(* Logix 5000 project; controller pracainz_ne 1769-L16ER-BB1B rev 30.11; software revision 30.00; part 2 of 2 *)
(* tags used below, declared in another part *)
   BELT_CONV_2_0 : ALIAS FOR BOOL_OUT_0;
   BELT_CONV_2_1 : ALIAS FOR BOOL_OUT_1;
   BELT_CONV_2_2 : ALIAS FOR BOOL_OUT_2;
   BELT_CONV_2_3 : ALIAS FOR BOOL_OUT_3;
   BELT_CONV_2_4 : ALIAS FOR BOOL_OUT_4;
   BELT_CONV_2_5 : ALIAS FOR BOOL_OUT_5;
   BELT_CONV_2_6 : ALIAS FOR BOOL_OUT_6;
   BELT_CONV_2_7 : ALIAS FOR BOOL_OUT_7;
   BELT_CONV_2_CCW : ALIAS FOR BOOL_OUT_27;
   BELT_CONV_4_0 : ALIAS FOR BOOL_OUT_8;
   BELT_CONV_4_1 : ALIAS FOR BOOL_OUT_9;
   BELT_CONV_4_2 : ALIAS FOR BOOL_OUT_10;
   BELT_CONV_4_3 : ALIAS FOR BOOL_OUT_11;
   BELT_CONV_CCW_0 : ALIAS FOR BOOL_OUT_23;
   BELT_CONV_CCW_3 : ALIAS FOR BOOL_OUT_24;
   BELT_CONV_CCW_4 : ALIAS FOR BOOL_OUT_25;
   BELT_CONV_CW_0 : ALIAS FOR BOOL_OUT_26;
   BELT_CONV_CW_1 : ALIAS FOR BOOL_OUT_20;
   BELT_CONV_CW_2 : ALIAS FOR BOOL_OUT_21;
   BELT_CONV_CW_5 : ALIAS FOR BOOL_OUT_22;
   CAP_SEN_0 : ALIAS FOR BOOL_IN_0;
   CAP_SEN_1 : ALIAS FOR BOOL_IN_1;
   CHAIN_0_LEFT : ALIAS FOR BOOL_OUT_16;
   CHAIN_0_N : ALIAS FOR BOOL_OUT_13;
   CHAIN_0_P : ALIAS FOR BOOL_OUT_12;
   CHAIN_0_RIGHT : ALIAS FOR BOOL_OUT_18;
   CHAIN_1_LEFT : ALIAS FOR BOOL_OUT_17;
   CHAIN_1_N : ALIAS FOR BOOL_OUT_15;
   CHAIN_1_P : ALIAS FOR BOOL_OUT_14;
   CHAIN_1_RIGHT : ALIAS FOR BOOL_OUT_19;
   COUNT : DINT;
   DIFF_SEN_0 : ALIAS FOR BOOL_IN_4;
   DIFF_SEN_1 : ALIAS FOR BOOL_IN_5;
   DIFF_SEN_2 : ALIAS FOR BOOL_IN_6;
   MANUAL : ALIAS FOR M_04;
   NOT_BLUE : ALIAS FOR M_24;
   NOT_GREEN : ALIAS FOR M_23;
   OSF_08_O : ALIAS FOR M_41;
   OSF_08_S : ALIAS FOR M_42;
   OSR_06_O : ALIAS FOR M_33;
   OSR_06_S : ALIAS FOR M_34;
   OSR_07_O : ALIAS FOR M_35;
   OSR_07_S : ALIAS FOR M_36;
   P_P_0_DETE : ALIAS FOR BOOL_IN_20;
   P_P_0_GRAB : ALIAS FOR BOOL_OUT_45;
   P_P_0_X : ALIAS FOR FLOAT_OUT_2;
   P_P_0_X_POSITION : ALIAS FOR FLOAT_IN_1;
   P_P_0_Y : ALIAS FOR FLOAT_OUT_0;
   P_P_0_Y_POSITION : ALIAS FOR FLOAT_IN_2;
   P_P_0_Z : ALIAS FOR FLOAT_OUT_4;
   P_P_0_Z_POSITION : ALIAS FOR FLOAT_IN_3;
   P_P_1_DETE : ALIAS FOR BOOL_IN_21;
   P_P_1_GRAB : ALIAS FOR BOOL_OUT_46;
   P_P_1_X : ALIAS FOR FLOAT_OUT_3;
   P_P_1_X_D : REAL;
   P_P_1_X_POSITION : ALIAS FOR FLOAT_IN_4;
   P_P_1_Y : ALIAS FOR FLOAT_OUT_1;
   P_P_1_Y_D : REAL;
   P_P_1_Y_POSITION : ALIAS FOR FLOAT_IN_5;
   P_P_1_Z : ALIAS FOR FLOAT_OUT_5;
   P_P_1_Z_D : REAL;
   P_P_1_Z_POSITION : ALIAS FOR FLOAT_IN_6;
   PUSH_0 : ALIAS FOR BOOL_OUT_47;
   PUSH_1 : ALIAS FOR BOOL_OUT_48;
   PUSHER_1 : BOOL;
   RETRO_SEN_0 : ALIAS FOR BOOL_IN_25;
   RETRO_SEN_3 : ALIAS FOR BOOL_IN_28;
   ROLL_4_0 : ALIAS FOR BOOL_OUT_50;
   ROLL_4_1 : ALIAS FOR BOOL_OUT_51;
   ROLL_4_2 : ALIAS FOR BOOL_OUT_52;
   ROLL_6_0 : ALIAS FOR BOOL_OUT_53;
   ROLL_6_1 : ALIAS FOR BOOL_OUT_54;
   TASMA_1 : BOOL;
   TASMA_2 : BOOL;
   TASMA_5 : BOOL;
   TASMA_9 : BOOL;
   auto_once : BOOL;
   BOOL_IN_41 : BOOL;
   BOOL_IN_43 : BOOL;
   BOOL_OUT_0 : BOOL;
   BOOL_OUT_1 : BOOL;
   BOOL_OUT_10 : BOOL;
   BOOL_OUT_11 : BOOL;
   BOOL_OUT_12 : BOOL;
   BOOL_OUT_13 : BOOL;
   BOOL_OUT_14 : BOOL;
   BOOL_OUT_15 : BOOL;
   BOOL_OUT_16 : BOOL;
   BOOL_OUT_17 : BOOL;
   BOOL_OUT_18 : BOOL;
   BOOL_OUT_19 : BOOL;
   BOOL_OUT_2 : BOOL;
   BOOL_OUT_20 : BOOL;
   BOOL_OUT_21 : BOOL;
   BOOL_OUT_22 : BOOL;
   BOOL_OUT_23 : BOOL;
   BOOL_OUT_24 : BOOL;
   BOOL_OUT_25 : BOOL;
   BOOL_OUT_26 : BOOL;
   BOOL_OUT_27 : BOOL;
   BOOL_OUT_29 : BOOL;
   BOOL_OUT_3 : BOOL;
   BOOL_OUT_30 : BOOL;
   BOOL_OUT_32 : BOOL;
   BOOL_OUT_33 : BOOL;
   BOOL_OUT_34 : BOOL;
   BOOL_OUT_35 : BOOL;
   BOOL_OUT_36 : BOOL;
   BOOL_OUT_37 : BOOL;
   BOOL_OUT_38 : BOOL;
   BOOL_OUT_39 : BOOL;
   BOOL_OUT_4 : BOOL;
   BOOL_OUT_40 : BOOL;
   BOOL_OUT_41 : BOOL;
   BOOL_OUT_42 : BOOL;
   BOOL_OUT_43 : BOOL;
   BOOL_OUT_44 : BOOL;
   BOOL_OUT_45 : BOOL;
   BOOL_OUT_46 : BOOL;
   BOOL_OUT_47 : BOOL;
   BOOL_OUT_48 : BOOL;
   BOOL_OUT_5 : BOOL;
   BOOL_OUT_50 : BOOL;
   BOOL_OUT_51 : BOOL;
   BOOL_OUT_52 : BOOL;
   BOOL_OUT_53 : BOOL;
   BOOL_OUT_54 : BOOL;
   BOOL_OUT_55 : BOOL;
   BOOL_OUT_56 : BOOL;
   BOOL_OUT_57 : BOOL;
   BOOL_OUT_6 : BOOL;
   BOOL_OUT_7 : BOOL;
   BOOL_OUT_8 : BOOL;
   BOOL_OUT_9 : BOOL;
   CHAIN_1_B : BOOL;
   CHAIN_1_F : BOOL;
   CHAIN_1_L : BOOL;
   CHAIN_1_R : BOOL;
   CHAIN_2_B : BOOL;
   CHAIN_2_F : BOOL;
   CHAIN_2_L : BOOL;
   CHAIN_2_R : BOOL;
   CLAMPED : BOOL;
   CLAMPED_R : BOOL;
   COUNT_R : DINT;
   EMERGENCY_ALL : BOOL;
   END_OF_DAY : BOOL;
   full_palet : BOOL;
   FULL_PALET_R : BOOL;
   Input_1 : BOOL;
   Input_1_R : BOOL;
   Input_2 : BOOL;
   Input_2_R : BOOL;
   Input_3 : BOOL;
   Input_3_R : BOOL;
   Input_4 : BOOL;
   Input_4_R : BOOL;
   Input_5 : BOOL;
   Input_5_R : BOOL;
   Input_6 : BOOL;
   Input_6_R : BOOL;
   Input_7 : BOOL;
   Input_7_R : BOOL;
   LEFT_PACK : BOOL;
   LEFT_PICK : BOOL;
   LEWA_LINIA : BOOL;
   LEWA_STRONA : BOOL;
   manual_once : BOOL;
   OSR_10_O : BOOL;
   OSR_10_S : BOOL;
   OSR_13_O : BOOL;
   OSR_14_O : BOOL;
   OSR_14_S : BOOL;
   P_P_0_X_D : REAL;
   P_P_0_Y_D : REAL;
   P_P_0_Z_D : REAL;
   PICK : BOOL;
   PRAWA_LINIA : BOOL;
   PRAWA_STRONA : BOOL;
   PUSHER_2 : BOOL;
   READY_L : BOOL;
   READY_R : BOOL;
   reset_timer : BOOL;
   reset_timer_l : BOOL;
   RIGHT_PACK : BOOL;
   RIGHT_PICK : BOOL;
   ROLL_1 : BOOL;
   ROLL_2 : BOOL;
   ROLL_3 : BOOL;
   ROLL_4 : BOOL;
   ROLL_5 : BOOL;
   ROLL_6 : BOOL;
   ROLL_7 : BOOL;
   START_ALL : BOOL;
   STOP_LEFT : BOOL;
   STOP_RIGHT : BOOL;
   stopped_left : BOOL;
   stopped_right : BOOL;
   TASMA_1_P : BOOL;
   TASMA_2_P : BOOL;
   TASMA_5_P : BOOL;
   TASMA_9_P : BOOL;
   TIMER_LEFT_P_P : TIMER;
   TIMER_RIGHT_P_P : TIMER;
   ton1 : TIMER;
   TON1_R : TIMER;
   ton2 : TIMER;
   TON2_R : TIMER;
   ton3 : TIMER;
   ton3_R : TIMER;
   ton4 : TIMER;
   TON4_R : TIMER;
   ton5 : TIMER;
   TON5_R : TIMER;
   ton6 : TIMER;
   TON6_R : TIMER;
   TON7 : TIMER;
   TON7_R : TIMER;
   X0 : REAL;
   X1 : REAL;
   Y0 : REAL;
   Y1 : REAL;
(* MainProgram, continued *)

ROUTINE R_07_timer_PICKNPLACE   (* ladder *)
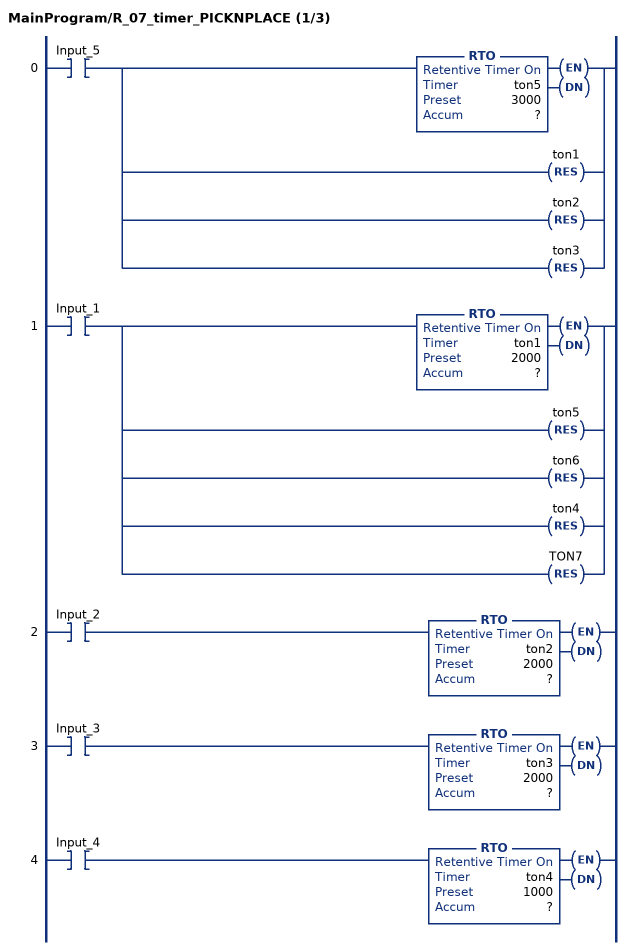
   0: XIC(Input_5)[RTO(ton5,?,?) ,RES(ton1) ,RES(ton2) ,RES(ton3) ];
   1: XIC(Input_1)[RTO(ton1,?,?) ,RES(ton5) ,RES(ton6) ,RES(ton4) ,RES(TON7) ];
   2: XIC(Input_2)RTO(ton2,?,?);
   3: XIC(Input_3)RTO(ton3,?,?);
   4: XIC(Input_4)RTO(ton4,?,?);
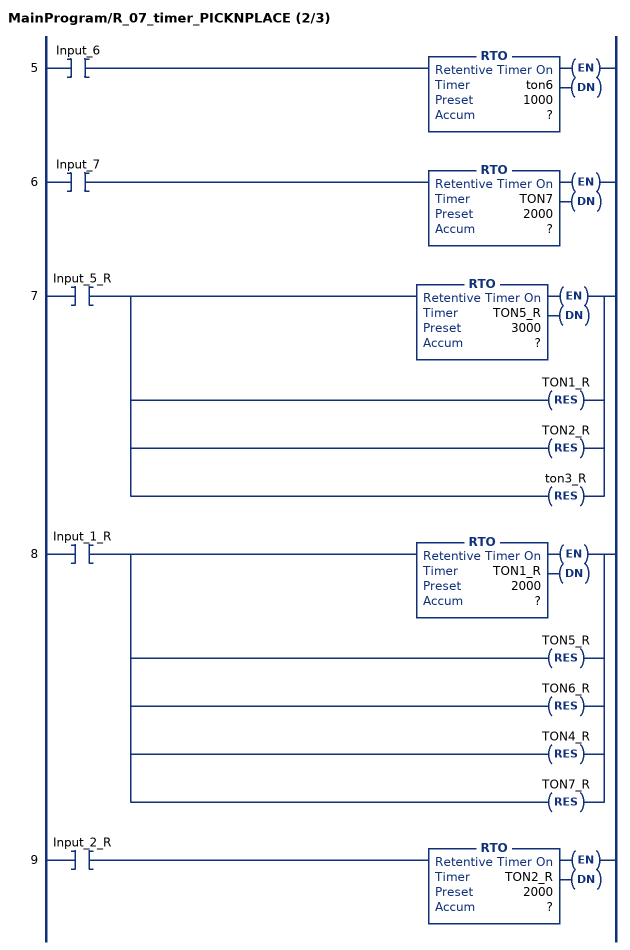
   5: XIC(Input_6)RTO(ton6,?,?);
   6: XIC(Input_7)RTO(TON7,?,?);
   7: XIC(Input_5_R)[RTO(TON5_R,?,?) ,RES(TON1_R) ,RES(TON2_R) ,RES(ton3_R) ];
   8: XIC(Input_1_R)[RTO(TON1_R,?,?) ,RES(TON5_R) ,RES(TON6_R) ,RES(TON4_R) ,RES(TON7_R) ];
   9: XIC(Input_2_R)RTO(TON2_R,?,?);
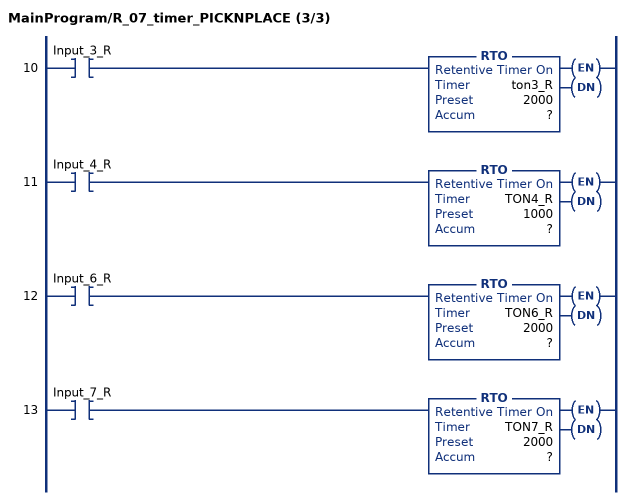
   10: XIC(Input_3_R)RTO(ton3_R,?,?);
   11: XIC(Input_4_R)RTO(TON4_R,?,?);
   12: XIC(Input_6_R)RTO(TON6_R,?,?);
   13: XIC(Input_7_R)RTO(TON7_R,?,?);
END_ROUTINE

ROUTINE R_08_Pick_and_Place_L   (* structured text *)
   IF LEFT_PACK THEN
   LEFT_PICK:=1;
   Input_1:=0;
   Input_2:=0;
   Input_3:=0;
   END_IF;
   
   IF  LEFT_PICK AND NOT(BOOL_IN_43) AND NOT(CLAMPED) AND (TIMER_LEFT_P_P.DN ) THEN  // ZACISKANIE
   BOOL_OUT_57:=1;
   END_IF;
   
   IF BOOL_IN_43 THEN
   CLAMPED:=1;
   BOOL_OUT_57:=0;
   P_P_1_Z:=0;
   Input_5:=1;
   END_IF;
   
   IF  LEFT_PICK AND CLAMPED THEN  // ZACZYNAMY OPERACJE RAMIENIEM
   LEFT_PICK:=0;
   END_IF;
   
   IF (Input_5)  THEN  // CHWYTANIE
   P_P_1_X:=9.1;
   P_P_1_Y:=6.5;
   IF ((P_P_1_X_POSITION=9.1) AND (P_P_1_Y_POSITION=6.5)) OR ton5.DN THEN
   P_P_1_Z:=8.5;
   IF (P_P_1_Z_POSITION>8.49 AND CLAMPED) then
   IF(P_P_1_DETE)THEN
   P_P_1_GRAB:=1;
   Input_6:=1;
   ELSE
   reset_timer_l:=1;
   CLAMPED:=0;
   END_IF;
   END_IF;
   END_IF;
   END_IF;
   
   
   IF  ton6.DN THEN
   P_P_1_Z:=0;
   Input_4:=1;
   IF ton4.DN THEN
   COUNT:=COUNT+1;
   READY_L:=1;
   LEFT_PICK:=0;
   END_IF;
   END_IF;
   
   
   
   
   IF READY_L AND NOT(full_palet) AND NOT(RETRO_SEN_0)  THEN
   
   CLAMPED:=0;
   Input_4:=0;
   Input_5:=0;
   Input_6:=0;
   Input_7:=0;
   
   CASE COUNT OF
   1:
   X1:=3.5;
   Y1:=6.8;
   
   2:
   X1:=5.29;
   Y1:=6.8;
   
   3:
   X1:=3.5;
   Y1:=3.8;
   
   4:
   X1:=5.29;
   Y1:=3.8;
   END_CASE;
   
   Input_1:=1;
   P_P_1_X:=X1;
   P_P_1_Y:=Y1;
   IF ((P_P_1_X_POSITION=X1) AND (P_P_1_Y_POSITION=Y1)) OR ton1.DN THEN
   P_P_1_Z:=8.5;
   Input_2:=1;
   IF (P_P_1_Z_POSITION>8.49) AND ton2.DN THEN
   P_P_1_GRAB:=0;
   P_P_1_Z:=5;
   READY_L:=0;
   END_IF;
   END_IF;
   END_IF;
   
   IF(COUNT=4) AND NOT(P_P_1_GRAB) THEN
   full_palet:=1;
   COUNT:=0;
   
   END_IF;
   
   
   
END_ROUTINE

ROUTINE R_08_Pick_and_Place_R   (* structured text *)
   IF RIGHT_PACK THEN
   RIGHT_PICK:=1;
   Input_1_R:=0;
   Input_2_R:=0;
   Input_3_R:=0;
   
   END_IF;
   
   IF  RIGHT_PICK AND NOT(BOOL_IN_41) AND NOT(CLAMPED_R) AND (TIMER_RIGHT_P_P.DN) THEN  // ZACISKANIE
   BOOL_OUT_55:=1;
   END_IF;
   
   IF BOOL_IN_41 THEN
   CLAMPED_R:=1;
   BOOL_OUT_55:=0;
   P_P_0_Z:=0;
   Input_5_R:=1;
   END_IF;
   
   IF  RIGHT_PICK AND CLAMPED_R THEN  // ZACZYNAMY OPERACJE RAMIENIEM
   RIGHT_PICK:=0;
   END_IF;
   
   IF (Input_5_R)  THEN  // CHWYTANIE
   P_P_0_X:=9.1;
   P_P_0_Y:=6.5;
   IF ((P_P_0_X_POSITION=9.1) AND (P_P_0_Y_POSITION=6.5)) OR TON5_R.DN THEN
   P_P_0_Z:=8.5;
   Input_7_R:=1;
   IF (P_P_0_Z_POSITION>8.49 AND CLAMPED_R) THEN
   IF(P_P_0_DETE)and TON7_R.DN THEN
   P_P_0_GRAB:=1;
   Input_6_R:=1;
   else
   reset_timer:=1;
   CLAMPED_R:=0;
   END_IF;
   END_IF;
   END_IF;
   END_IF;
   
   
   
   IF  TON6_R.DN THEN
   P_P_0_Z:=0;
   Input_4_R:=1;
   IF TON4_R.DN THEN
   COUNT_R:=COUNT_R+1;
   READY_R:=1;
   RIGHT_PICK:=0;
   END_IF;
   END_IF;
   
   
   
   IF READY_R AND NOT(FULL_PALET_R) AND NOT(RETRO_SEN_3)  THEN
   CLAMPED_R:=0;
   Input_4_R:=0;
   Input_5_R:=0;
   Input_6_R:=0;
   Input_7_R:=0;
   
   CASE COUNT_R OF
   1:
   X0:=3.5;
   Y0:=6.0;
   
   2:
   X0:=5.3;
   Y0:=6.0;
   
   3:
   X0:=3.5;
   Y0:=2.9;
   
   4:
   X0:=5.3;
   Y0:=2.9;
   END_CASE;
   
   Input_1_R:=1;
   P_P_0_X:=X0;
   P_P_0_Y:=Y0;
   IF ((P_P_0_X_POSITION=X0) AND (P_P_0_Y_POSITION=Y0)) OR TON1_R.DN THEN
   P_P_0_Z:=8.5;
   Input_2_R:=1;
   IF (P_P_0_Z_POSITION>8.49) AND TON2_R.DN THEN
   P_P_0_GRAB:=0;
   P_P_0_Z:=5;
   READY_R:=0;
   END_IF;
   END_IF;
   END_IF;
   
   IF(COUNT_R=4) AND NOT(P_P_0_GRAB) THEN
   FULL_PALET_R:=1;
   COUNT_R:=0;
   
   END_IF;
   
   
   
END_ROUTINE

ROUTINE R_09_roller_n_chain   (* ladder *)
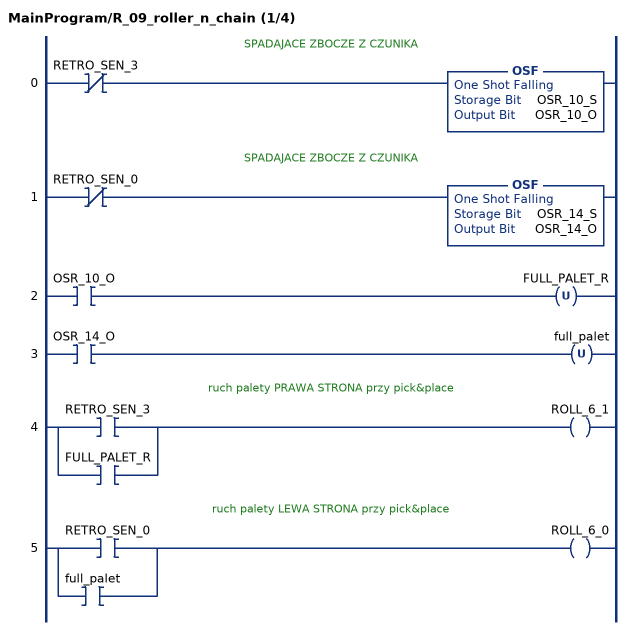
   // SPADAJACE ZBOCZE Z CZUNIKA
   0: XIO(RETRO_SEN_3)OSF(OSR_10_S,OSR_10_O);
   // SPADAJACE ZBOCZE Z CZUNIKA
   1: XIO(RETRO_SEN_0)OSF(OSR_14_S,OSR_14_O);
   2: XIC(OSR_10_O)OTU(FULL_PALET_R);
   3: XIC(OSR_14_O)OTU(full_palet);
   // ruch palety PRAWA STRONA przy pick&place
   4: [XIC(RETRO_SEN_3) ,XIC(FULL_PALET_R) ]OTE(ROLL_6_1);
   // ruch palety LEWA STRONA przy pick&place
   5: [XIC(RETRO_SEN_0) ,XIC(full_palet) ]OTE(ROLL_6_0);
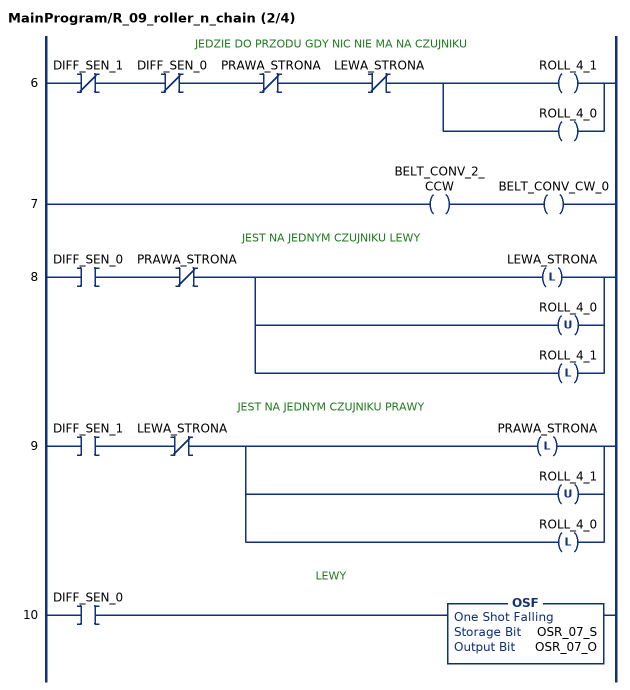
   // JEDZIE DO PRZODU GDY NIC NIE MA NA CZUJNIKU
   6: XIO(DIFF_SEN_1)XIO(DIFF_SEN_0)XIO(PRAWA_STRONA)XIO(LEWA_STRONA)[OTE(ROLL_4_1) ,OTE(ROLL_4_0) ];
   7: OTE(BELT_CONV_2_CCW)OTE(BELT_CONV_CW_0);
   // JEST NA JEDNYM CZUJNIKU LEWY
   8: XIC(DIFF_SEN_0)XIO(PRAWA_STRONA)[OTL(LEWA_STRONA) ,OTU(ROLL_4_0) ,OTL(ROLL_4_1) ];
   // JEST NA JEDNYM CZUJNIKU PRAWY
   9: XIC(DIFF_SEN_1)XIO(LEWA_STRONA)[OTL(PRAWA_STRONA) ,OTU(ROLL_4_1) ,OTL(ROLL_4_0) ];
   // LEWY
   10: XIC(DIFF_SEN_0)OSF(OSR_07_S,OSR_07_O);
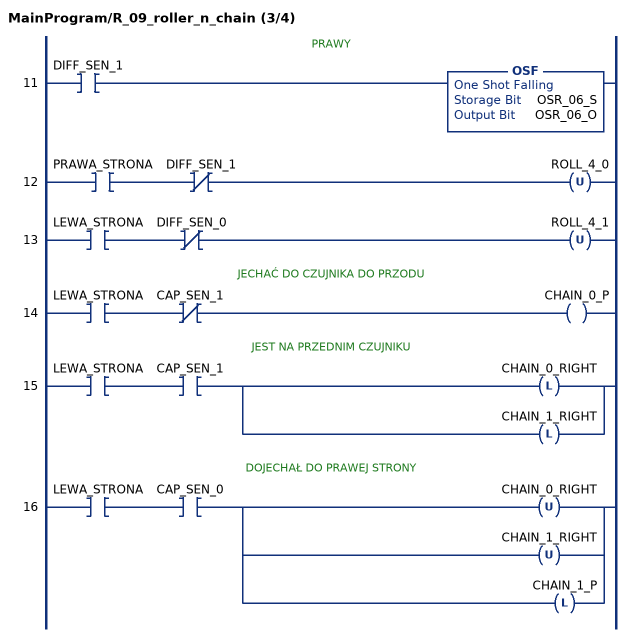
   // PRAWY
   11: XIC(DIFF_SEN_1)OSF(OSR_06_S,OSR_06_O);
   12: XIC(PRAWA_STRONA)XIO(DIFF_SEN_1)OTU(ROLL_4_0);
   13: XIC(LEWA_STRONA)XIO(DIFF_SEN_0)OTU(ROLL_4_1);
   // JECHAĆ DO CZUJNIKA DO PRZODU
   14: XIC(LEWA_STRONA)XIO(CAP_SEN_1)OTE(CHAIN_0_P);
   // JEST NA PRZEDNIM CZUJNIKU
   15: XIC(LEWA_STRONA)XIC(CAP_SEN_1)[OTL(CHAIN_0_RIGHT) ,OTL(CHAIN_1_RIGHT) ];
   // DOJECHAŁ DO PRAWEJ STRONY
   16: XIC(LEWA_STRONA)XIC(CAP_SEN_0)[OTU(CHAIN_0_RIGHT) ,OTU(CHAIN_1_RIGHT) ,OTL(CHAIN_1_P) ];
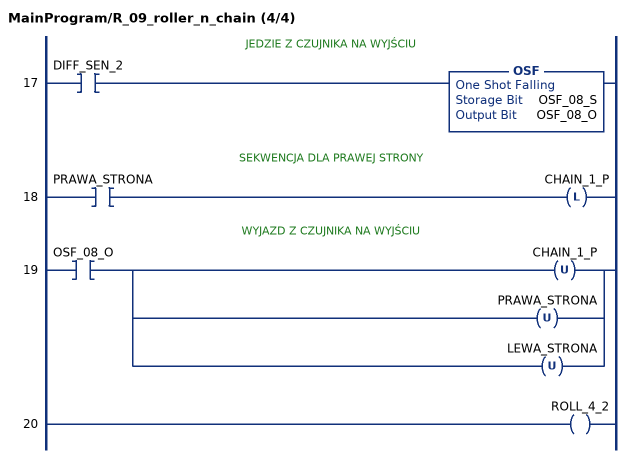
   // JEDZIE Z CZUJNIKA NA WYJŚCIU
   17: XIC(DIFF_SEN_2)OSF(OSF_08_S,OSF_08_O);
   // SEKWENCJA DLA PRAWEJ STRONY
   18: XIC(PRAWA_STRONA)OTL(CHAIN_1_P);
   // WYJAZD Z CZUJNIKA NA WYJŚCIU
   19: XIC(OSF_08_O)[OTU(CHAIN_1_P) ,OTU(PRAWA_STRONA) ,OTU(LEWA_STRONA) ];
   20: OTE(ROLL_4_2);
END_ROUTINE

ROUTINE R_10_MANUAL   (* ladder *)
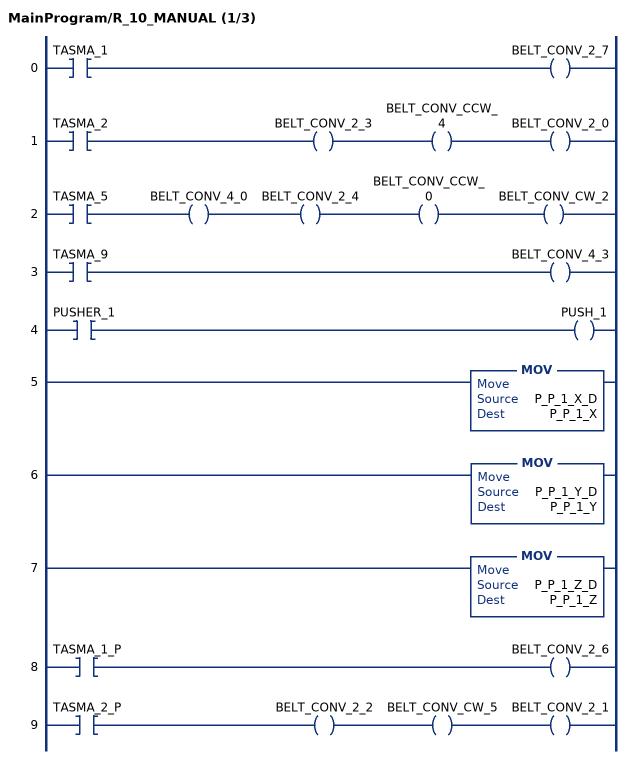
   0: XIC(TASMA_1)OTE(BELT_CONV_2_7);
   1: XIC(TASMA_2)OTE(BELT_CONV_2_3)OTE(BELT_CONV_CCW_4)OTE(BELT_CONV_2_0);
   2: XIC(TASMA_5)OTE(BELT_CONV_4_0)OTE(BELT_CONV_2_4)OTE(BELT_CONV_CCW_0)OTE(BELT_CONV_CW_2);
   3: XIC(TASMA_9)OTE(BELT_CONV_4_3);
   4: XIC(PUSHER_1)OTE(PUSH_1);
   5: MOV(P_P_1_X_D,P_P_1_X);
   6: MOV(P_P_1_Y_D,P_P_1_Y);
   7: MOV(P_P_1_Z_D,P_P_1_Z);
   8: XIC(TASMA_1_P)OTE(BELT_CONV_2_6);
   9: XIC(TASMA_2_P)OTE(BELT_CONV_2_2)OTE(BELT_CONV_CW_5)OTE(BELT_CONV_2_1);
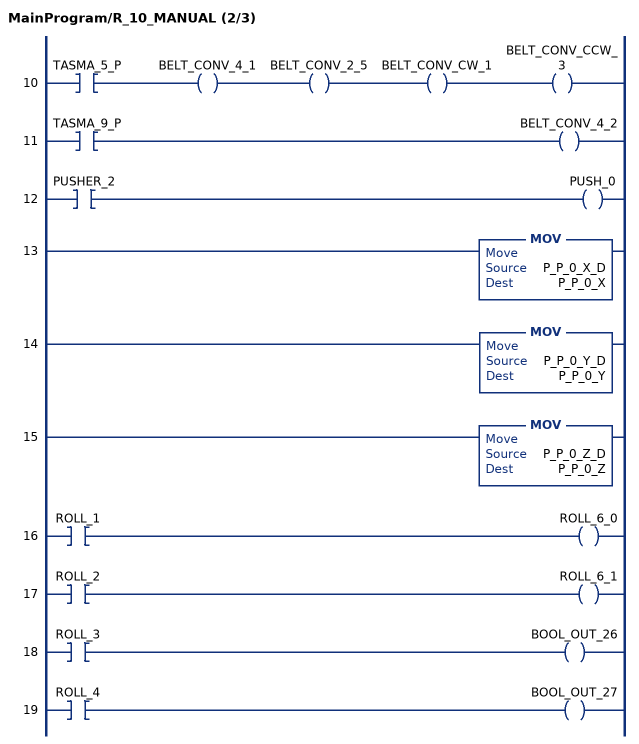
   10: XIC(TASMA_5_P)OTE(BELT_CONV_4_1)OTE(BELT_CONV_2_5)OTE(BELT_CONV_CW_1)OTE(BELT_CONV_CCW_3);
   11: XIC(TASMA_9_P)OTE(BELT_CONV_4_2);
   12: XIC(PUSHER_2)OTE(PUSH_0);
   13: MOV(P_P_0_X_D,P_P_0_X);
   14: MOV(P_P_0_Y_D,P_P_0_Y);
   15: MOV(P_P_0_Z_D,P_P_0_Z);
   16: XIC(ROLL_1)OTE(ROLL_6_0);
   17: XIC(ROLL_2)OTE(ROLL_6_1);
   18: XIC(ROLL_3)OTE(BOOL_OUT_26);
   19: XIC(ROLL_4)OTE(BOOL_OUT_27);
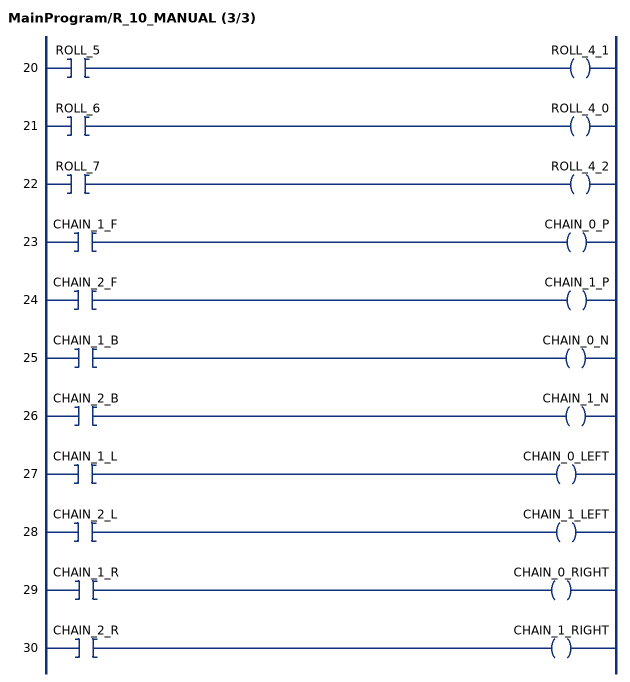
   20: XIC(ROLL_5)OTE(ROLL_4_1);
   21: XIC(ROLL_6)OTE(ROLL_4_0);
   22: XIC(ROLL_7)OTE(ROLL_4_2);
   23: XIC(CHAIN_1_F)OTE(CHAIN_0_P);
   24: XIC(CHAIN_2_F)OTE(CHAIN_1_P);
   25: XIC(CHAIN_1_B)OTE(CHAIN_0_N);
   26: XIC(CHAIN_2_B)OTE(CHAIN_1_N);
   27: XIC(CHAIN_1_L)OTE(CHAIN_0_LEFT);
   28: XIC(CHAIN_2_L)OTE(CHAIN_1_LEFT);
   29: XIC(CHAIN_1_R)OTE(CHAIN_0_RIGHT);
   30: XIC(CHAIN_2_R)OTE(CHAIN_1_RIGHT);
END_ROUTINE

ROUTINE R_11_RESET   (* structured text *)
   IF auto_once OR manual_once OR EMERGENCY_ALL THEN
   LEWA_LINIA:=0;
   PRAWA_LINIA:=0;
   STOP_LEFT:=0;
   STOP_RIGHT:=0;
   stopped_left:=0;
   stopped_right:=0;
   NOT_BLUE:=0;
   NOT_GREEN:=0;
   PUSH_0:=0;
   PUSH_1:=0;
   full_palet:=0;
   FULL_PALET_R:=0;
   COUNT:=0;
   COUNT_R:=0;
   LEWA_STRONA:=0;
   PRAWA_STRONA:=0;
   CLAMPED:=0;
   CLAMPED_R:=0;
   LEFT_PICK:=0;
   RIGHT_PICK:=0;
   LEFT_PACK:=0;
   RIGHT_PACK:=0;
   READY_L:=0;
   READY_R:=0;
   Input_1:=0;
   Input_2:=0;
   Input_3:=0;
   Input_4:=0;
   Input_5:=0;
   Input_6:=0;
   Input_1_R:=0;
   Input_2_R:=0;
   Input_3_R:=0;
   Input_4_R:=0;
   Input_5_R:=0;
   Input_6_R:=0;
   If auto_once then
   P_P_1_Z:=0;
   P_P_0_Z:=0;
   auto_once:=0;
   end_if;
   end_if;
   
   if not(MANUAL) then
   TASMA_1:=0;
   TASMA_2:=0;
   TASMA_5:=0;
   TASMA_9:=0;
   PUSHER_1:=0;
   TASMA_1_P:=0;
   TASMA_2_P:=0;
   TASMA_5_P:=0;
   TASMA_9_P:=0;
   PUSHER_2:=0;
   ROLL_1:=0;
   ROLL_2:=0;
   ROLL_3:=0;
   ROLL_4:=0;
   ROLL_5:=0;
   ROLL_6:=0;
   ROLL_7:=0;
   CHAIN_1_F:=0;
   CHAIN_2_F:=0;
   CHAIN_1_B:=0;
   CHAIN_2_B:=0;
   CHAIN_1_L:=0;
   CHAIN_2_L:=0;
   CHAIN_1_R:=0;
   CHAIN_2_R:=0;
   
   end_if;
   
   
   IF  START_ALL OR END_OF_DAY then
   BOOL_OUT_35:=0;
   BOOL_OUT_36:=0;
   END_IF;
   
    IF (OSR_13_O) and not(COUNT=0) THEN
    full_palet:=1;
    END_IF;
   
    IF (OSR_13_O) and not(COUNT_R=0) THEN
   FULL_PALET_R:=1;
    END_IF;
   
   
END_ROUTINE

ROUTINE R_12_EMERGENCY   (* structured text *)
   P_P_1_Z:=P_P_1_Z_POSITION;
   P_P_1_Y:=P_P_1_Y_POSITION;
   P_P_1_X:=P_P_1_X_POSITION;
   P_P_0_Z:=P_P_0_Z_POSITION;
   P_P_0_Y:=P_P_0_Y_POSITION;
   P_P_0_X:=P_P_0_X_POSITION;
   BOOL_OUT_0:=0;
   BOOL_OUT_1:=0;
   BOOL_OUT_2:=0;
   BOOL_OUT_3:=0;
   BOOL_OUT_4:=0;
   BOOL_OUT_5:=0;
   BOOL_OUT_6:=0;
   BOOL_OUT_7:=0;
   BOOL_OUT_8:=0;
   BOOL_OUT_9:=0;
   BOOL_OUT_10:=0;
   BOOL_OUT_11:=0;
   BOOL_OUT_12:=0;
   BOOL_OUT_13:=0;
   BOOL_OUT_14:=0;
   BOOL_OUT_15:=0;
   BOOL_OUT_16:=0;
   BOOL_OUT_17:=0;
   BOOL_OUT_18:=0;
   BOOL_OUT_19:=0;
   BOOL_OUT_20:=0;
   BOOL_OUT_21:=0;
   BOOL_OUT_22:=0;
   BOOL_OUT_23:=0;
   BOOL_OUT_24:=0;
   BOOL_OUT_25:=0;
   BOOL_OUT_26:=0;
   BOOL_OUT_27:=0;
   BOOL_OUT_29:=0;
   BOOL_OUT_30:=0;
   BOOL_OUT_32:=0;
   BOOL_OUT_33:=0;
   BOOL_OUT_34:=0;
   BOOL_OUT_35:=1;
   BOOL_OUT_36:=1;
   BOOL_OUT_37:=0;
   BOOL_OUT_38:=0;
   BOOL_OUT_39:=0;
   BOOL_OUT_40:=0;
   BOOL_OUT_41:=0;
   BOOL_OUT_42:=0;
   BOOL_OUT_43:=0;
   BOOL_OUT_44:=0;
   BOOL_OUT_45:=0;
   BOOL_OUT_46:=0;
   BOOL_OUT_47:=0;
   BOOL_OUT_48:=0;
   BOOL_OUT_50:=0;
   BOOL_OUT_51:=0;
   BOOL_OUT_52:=0;
   BOOL_OUT_53:=0;
   BOOL_OUT_54:=0;
   BOOL_OUT_55:=0;
   BOOL_OUT_56:=0;
   BOOL_OUT_57:=0;
   TASMA_1:=0;
   TASMA_2:=0;
   TASMA_5:=0;
   TASMA_9:=0;
   PUSHER_1:=0;
   TASMA_1_P:=0;
   TASMA_2_P:=0;
   TASMA_5_P:=0;
   TASMA_9_P:=0;
   PUSHER_2:=0;
   manual_once:=0;
   
   
   
   
   
   
   
   
END_ROUTINE
END_PROGRAM
